FUNCTION_BLOCK NE (* IEC 61131-3,Table 28#10 *)
  (* Standard: IEC 61131-3; Classification: Comparison *)
  (* Version 0.1, 2001-10-05, JHC, Rockwell Automation, Copied/modified to use ANY.equals(). *)
  (* Version 0.0, 1998-12-22, JHC, Rockwell Automation, NE_INT.src version *)
  (* Compiler header: package fb.rt.plc.comp;import fb.rt.plc.*; *)
  (* Compiler classdef: class NE extends FBR1131Function2 *)
  (* Compiler Java IBM VisualAge 3.0 *)
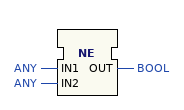
  VAR_INPUT
    IN1 : ANY;
    IN2 : ANY;
  END_VAR
  VAR_OUTPUT
    OUT : BOOL;
  END_VAR
END_FUNCTION_BLOCK
